FUNCTION_BLOCK LiftControl (* Basic Function Block Type *)
  (* Standard: 61499-2 *)
  (* Version 0.0, 1/14/2024, midxav, Template *)
  PACKAGE Main;
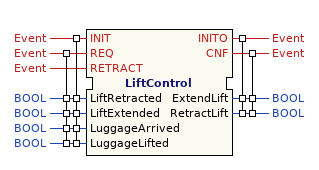
  EVENT_INPUT
    INIT WITH LiftRetracted, LiftExtended, LuggageArrived, LuggageLifted; (* Initialization Request *)
    REQ WITH LiftRetracted, LiftExtended, LuggageArrived, LuggageLifted; (* Normal Execution Request *)
    RETRACT;
  END_EVENT
  EVENT_OUTPUT
    INITO WITH ExtendLift, RetractLift; (* Initialization Confirm *)
    CNF WITH ExtendLift, RetractLift; (* Execution Confirmation *)
  END_EVENT
  VAR_INPUT
    LiftRetracted : BOOL; (* Input event qualifier *)
    LiftExtended : BOOL;
    LuggageArrived : BOOL;
    LuggageLifted : BOOL;
  END_VAR
  VAR_OUTPUT
    ExtendLift : BOOL; (* Output event qualifier *)
    RetractLift : BOOL;
  END_VAR
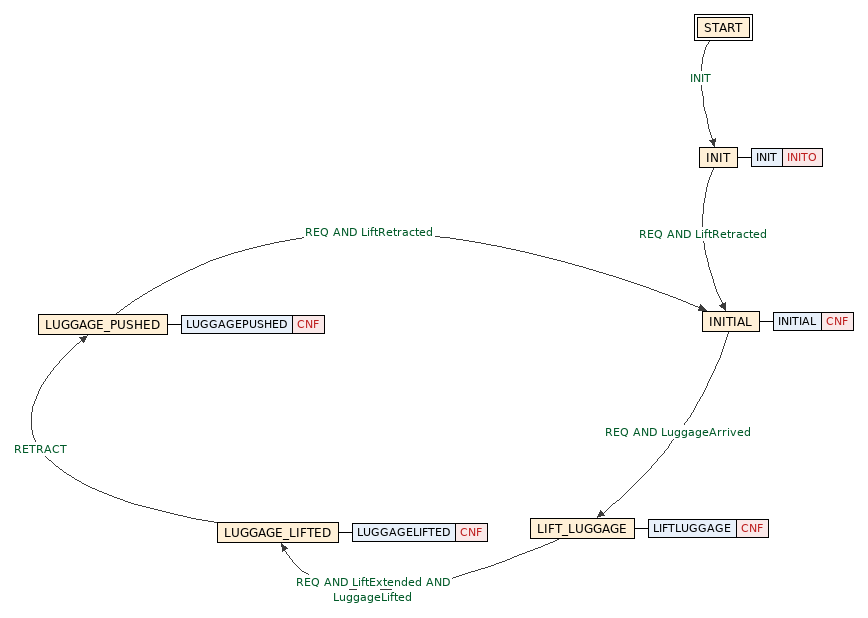
  EC_STATES
    START; (* Initial State *)
    INIT : INIT -> INITO; (* Initialization *)
    INITIAL : INITIAL -> CNF;
    LIFT_LUGGAGE : LIFTLUGGAGE -> CNF;
    LUGGAGE_LIFTED : LUGGAGELIFTED -> CNF;
    LUGGAGE_PUSHED : LUGGAGEPUSHED -> CNF;
  END_STATES
  EC_TRANSITIONS
    START TO INIT := INIT;
    INIT TO INITIAL := REQ AND LiftRetracted;
    INITIAL TO LIFT_LUGGAGE := REQ AND LuggageArrived;
    LIFT_LUGGAGE TO LUGGAGE_LIFTED := REQ AND LiftExtended AND LuggageLifted;
    LUGGAGE_LIFTED TO LUGGAGE_PUSHED := RETRACT;
    LUGGAGE_PUSHED TO INITIAL := REQ AND LiftRetracted;
  END_TRANSITIONS
  ALGORITHM INIT IN ST:
ExtendLift:= FALSE;
RetractLift:=TRUE;
  END_ALGORITHM
  ALGORITHM INITIAL IN ST:
RetractLift:=FALSE;
  END_ALGORITHM
  ALGORITHM LIFTLUGGAGE IN ST:
ExtendLift:=TRUE;
  END_ALGORITHM
  ALGORITHM LUGGAGELIFTED IN ST:
ExtendLift:=FALSE;
  END_ALGORITHM
  ALGORITHM LUGGAGEPUSHED IN ST:
RetractLift:=TRUE;
  END_ALGORITHM
END_FUNCTION_BLOCK
